(********************* G.D S.p.A. - Technical Department ***********************************
This program has been generated automatically from Application Designer DE&F
********************************************************************************************)
PROGRAM dbg_csp_case_tr_accu_ls_width
VAR
  axis_shd : axis_shadow;
END_VAR

_objects_manager();

IF	g_application_status <> APPLICATION_STATUS_RUNNING
THEN
	RETURN;
END_IF

CASE process_get_mode(CONVERSION_this := dbg_root.prc) OF
	MODE_ABSENT,
	MODE_INACTIVE:
		RETURN;
	MODE_TEST:
		RETURN;
END_CASE

ACTION _objects_manager:
IF	objects_initialization()
THEN
	axis_shadow_init(
		sim_mode:= SHADOW_SIMULATION_MODE_AUTOMATIC, 
		father:= csp_case_tr_accu_ls_width.axis, 
		process:= dbg_root.prc, 
		CONVERSION_this:= axis_shd);

	RETURN;
END_IF

IF	objects_running()
THEN
	axis_shadow_cycle(axis_shd);
END_IF
END_ACTION

END_PROGRAM

(* stored: Version 1.1.0.1, ProductVersion 3.1.4022.12
   POU dbg_csp_case_tr_accu_ls_width: Id {f8e02f3d-90ec-4f9f-b18f-602cb00ec77d}, SpecialFunc None
   Action _objects_manager: Id {bbc799aa-e401-4fda-90ae-7c8673ebc70b} *)
